(* Logix 5000 project; controller cal1615 1756-L62 rev 16.20; software revision 16.05; part 46 of 78 *)
(* tags used below, declared in another part *)
   FAULT : BOOL;   // Fault AFI
   HMI : BOOL;   // AFI HMI
   p01r02 : routine;   // System Misc Control
   p01r09_pb_global_reset : BOOL;   // System Modes PB: Global Fault Reset
   p01r09_stretch_mode : BOOL;
   p22_ai_amps : REAL;   // Tension Stand 1 Analog Input Tension Stand 1 Motor Current
   p22_ai_hz : REAL;   // Tension Stand 1 Analog Input Tension Stand 1 Motor Hertz
   p22_ai_speed : REAL;
   p22_ai_torque : REAL;
   p22_ai_ts1_lc : REAL;   // Tension Stand 1 Analog Input Loadcell
   p22_ao_selected_speed : REAL;   // Tension Stand 1 VFD Selected Speed
   p22_ao_torque : REAL;
   p22_ao_vfd : REAL;
   p22_control_word : INT;
   p22_di_brake : BOOL;   // Tension Stand 1 Digital Input Brake Temperature OK
   p22_di_close_nip_roll : BOOL;   // Tension Stand 1 Digital Input SS: Close Nip Roll
   p22_di_jog : BOOL;   // Tension Stand 1 Digital Input SS: Jog
   p22_di_jog_fwd : BOOL;   // Tension Stand 1 Digital Input PB: Jog Forward
   p22_di_jog_rev : BOOL;   // Tension Stand 1 Digital Input PB: Jog Reverse
   p22_di_open_nip_roll : BOOL;   // Tension Stand 1 Digital Input SS: Open Nip Roll
   p22_di_run : BOOL;   // Tension Stand 1 Digital Input SS: Run
   p22_di_therm : BOOL;   // Tension Stand 1 Digital Input Motor Temperature OK
   p22_dint_to_hmi : DINT[16];   // Tension Stand 1 Dint to HMI
   p22_do_close_nip_roll : BOOL;   // Tension Stand 1 Digital Output Close Tension Stand 1 Nip Roll
   p22_status_word : INT;
   p22_ts1_gear_ratio : REAL;
   p22_ts1_roll_diameter_ft : REAL;
   p22_vfd_input_max : REAL;
   p22_vfd_input_min : REAL;
   p22_vfd_output_max : REAL;
   p22_vfd_output_min : REAL;
   p22r01 : routine;   // Tension Stand 1 Main
   p22r03 : routine;   // Tension Stand 1 Input
   p22r03_ave_tq : REAL;
   p22r03_hz : SYS_SCP;   // Tension Stand 1 Analog Inputs SCP Hz
   p22r03_lc_input_max : REAL;
   p22r03_lc_input_min : REAL;
   p22r03_lc_output_max : REAL;
   p22r03_lc_output_min : REAL;
   p22r03_lc_scp : SYS_SCP;   // Tension Stand 1 Analog Input Load Cell Scaling
   p22r03_sample_timer : TIMER;
   p22r03_scaled_vfd_in : REAL;
   p22r03_timer_fault : TIMER[4];   // Tension Stand 1 Input Fault Delay
   p22r03_timer_warning : TIMER[4];   // Tension Stand 1 Input Warning Delay
   p22r03_tq_ave_ctrl : CONTROL;
   p22r03_tq_buffer : REAL[20];
   p22r03_tq_fifo : CONTROL;
   p22R03_ts1_vfd_rpm_to_speed : SYS_RPM_TO_SPEED;   // Tension Stand 1 Analog Input VFD RPM to Roll Surface Speed
   p22r03_unload : DINT;
   p22r03_vfd_in_scaling : SYS_SCP;
   p22r03_vfd_input_max : REAL;
   p22r03_vfd_input_min : REAL;
   p22r03_vfd_out_scaling : SYS_SCP;
   p22r03_vfd_output_max : REAL;
   p22r03_vfd_output_min : REAL;
   p22r04 : routine;   // Tension Stand 1 Output
   p22r04_speed_to_vfd_1 : SYS_SPEED_TO_VFD;   // Tension Stand 1 Analog Output Speed to VFD
   p22r04_timer_fault : TIMER[4];   // Tension Stand 1 Output Fault Delay
   p22r04_timer_warning : TIMER[4];   // Tension Stand 1 Output Warning Delay
   p22r05 : routine;   // Tension Stand 1 Dint to HMI
   p22r05_timer_fault : TIMER[4];   // Tension Stand 1 Dint to HMI Fault Delay
   p22r05_timer_warning : TIMER[4];   // Tension Stand 1 Dint to HMI Warning Delay
   p22r09_mode_jog : BOOL;   // Tension Stand 1 Modes Jog Mode
   p22r09_mode_run : BOOL;   // Tension Stand 1 Modes Run Mode
   p22r09_mode_thread : BOOL;   // Tension Stand 1 Modes Thread Mode
   p25r03 : routine;
(* P22_Tension_Stand_1, continued *)

ROUTINE R03_Input   (* ladder *)
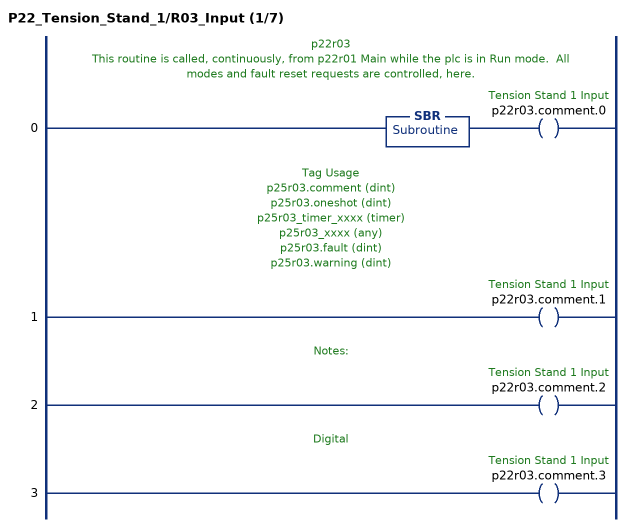
   // p22r03
   // This routine is called, continuously, from p22r01 Main while the plc is in Run mode.  All modes and fault reset requests are controlled, here.
   0: SBR()OTE(p22r03.comment.0);
   // Tag Usage
   // p25r03.comment (dint)
   // p25r03.oneshot (dint)
   // p25r03_timer_xxxx (timer)
   // p25r03_xxxx (any)
   // p25r03.fault (dint)
   // p25r03.warning (dint)
   1: OTE(p22r03.comment.1);
   // Notes:
   2: OTE(p22r03.comment.2);
   // Digital
   3: OTE(p22r03.comment.3);
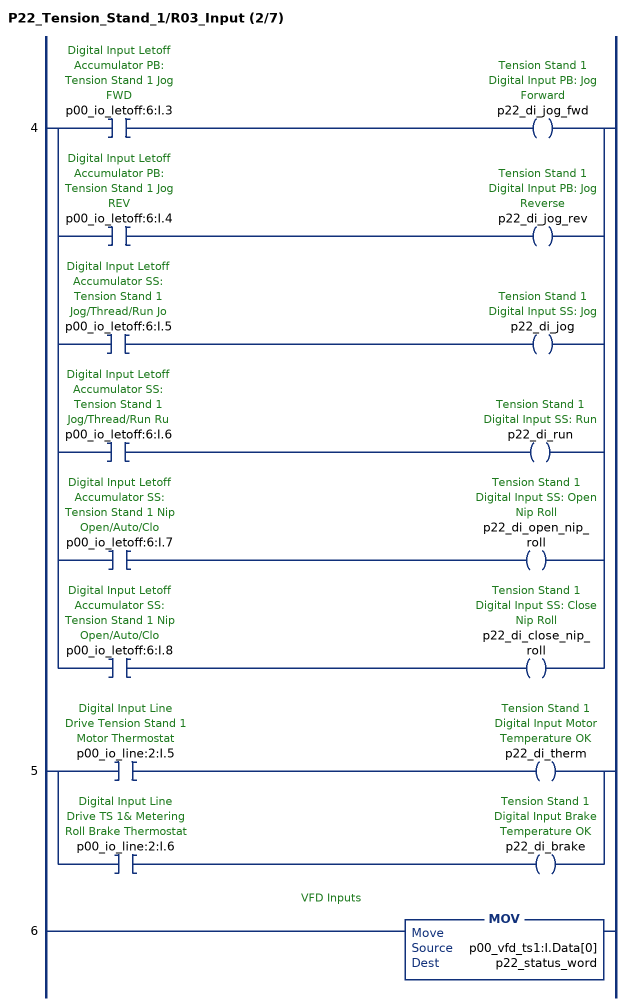
   4: [XIC(p00_io_letoff:6:I.3) OTE(p22_di_jog_fwd) ,XIC(p00_io_letoff:6:I.4) OTE(p22_di_jog_rev) ,XIC(p00_io_letoff:6:I.5) OTE(p22_di_jog) ,XIC(p00_io_letoff:6:I.6) OTE(p22_di_run) ,XIC(p00_io_letoff:6:I.7) OTE(p22_di_open_nip_roll) ,XIC(p00_io_letoff:6:I.8) OTE(p22_di_close_nip_roll) ];
   5: [XIC(p00_io_line:2:I.5) OTE(p22_di_therm) ,XIC(p00_io_line:2:I.6) OTE(p22_di_brake) ];
   // VFD Inputs
   6: MOV(p00_vfd_ts1:I.Data[0],p22_status_word);
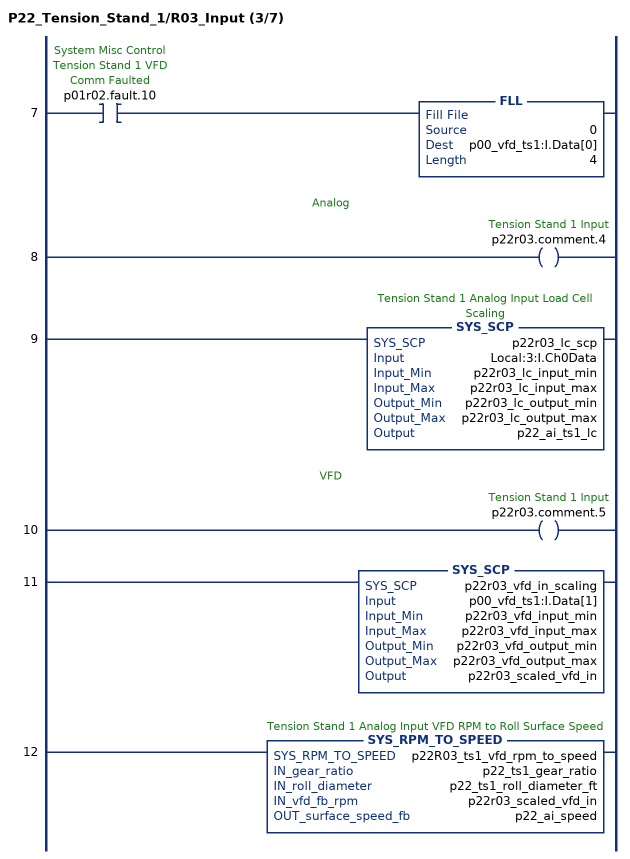
   7: XIC(p01r02.fault.10)FLL(0,p00_vfd_ts1:I.Data[0],4);
   // Analog
   8: OTE(p22r03.comment.4);
   9: SYS_SCP(p22r03_lc_scp,Local:3:I.Ch0Data,p22r03_lc_input_min,p22r03_lc_input_max,p22r03_lc_output_min,p22r03_lc_output_max,p22_ai_ts1_lc);
   // VFD
   10: OTE(p22r03.comment.5);
   11: SYS_SCP(p22r03_vfd_in_scaling,p00_vfd_ts1:I.Data[1],p22r03_vfd_input_min,p22r03_vfd_input_max,p22r03_vfd_output_min,p22r03_vfd_output_max,p22r03_scaled_vfd_in);
   12: SYS_RPM_TO_SPEED(p22R03_ts1_vfd_rpm_to_speed,p22_ts1_gear_ratio,p22_ts1_roll_diameter_ft,p22r03_scaled_vfd_in,p22_ai_speed);
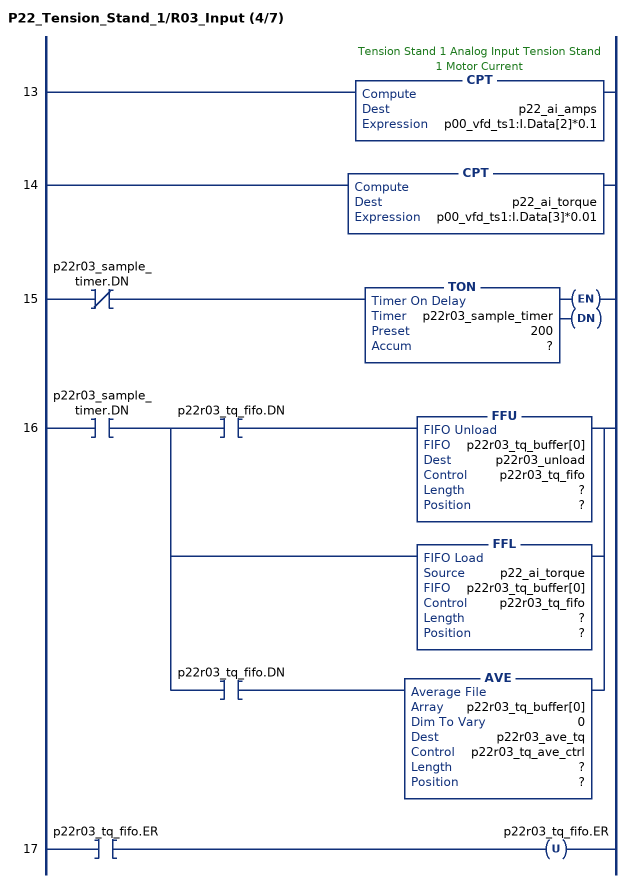
   13: CPT(p22_ai_amps,p00_vfd_ts1:I.Data[2]*0.1);
   14: CPT(p22_ai_torque,p00_vfd_ts1:I.Data[3]*0.01);
   15: XIO(p22r03_sample_timer.DN)TON(p22r03_sample_timer,?,?);
   16: XIC(p22r03_sample_timer.DN)[XIC(p22r03_tq_fifo.DN) FFU(p22r03_tq_buffer[0],p22r03_unload,p22r03_tq_fifo,?,?) ,FFL(p22_ai_torque,p22r03_tq_buffer[0],p22r03_tq_fifo,?,?) ,XIC(p22r03_tq_fifo.DN) AVE(p22r03_tq_buffer[0],0,p22r03_ave_tq,p22r03_tq_ave_ctrl,?,?) ];
   17: XIC(p22r03_tq_fifo.ER)OTU(p22r03_tq_fifo.ER);
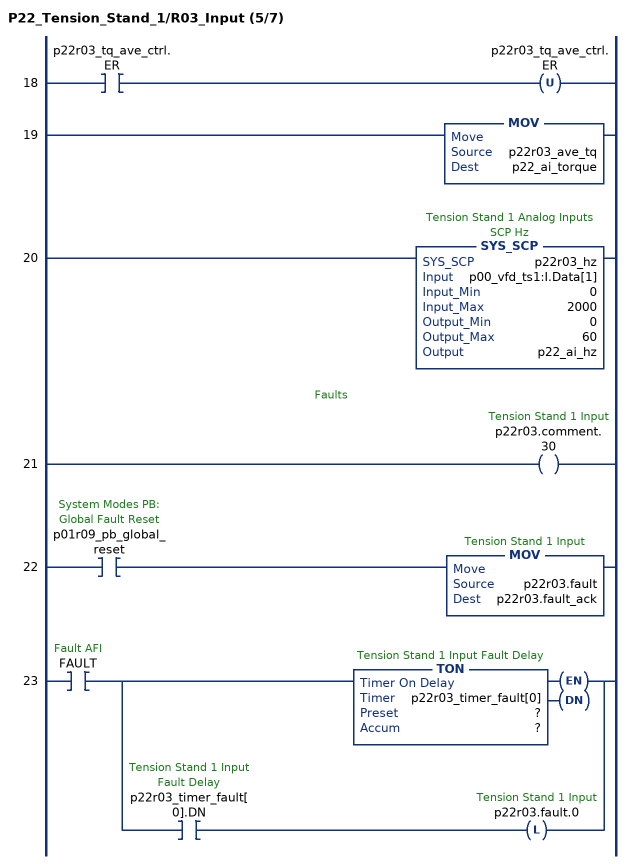
   18: XIC(p22r03_tq_ave_ctrl.ER)OTU(p22r03_tq_ave_ctrl.ER);
   19: MOV(p22r03_ave_tq,p22_ai_torque);
   20: SYS_SCP(p22r03_hz,p00_vfd_ts1:I.Data[1],0,2000,0,60,p22_ai_hz);
   // Faults
   21: OTE(p22r03.comment.30);
   22: XIC(p01r09_pb_global_reset)MOV(p22r03.fault,p22r03.fault_ack);
   23: XIC(FAULT)[TON(p22r03_timer_fault[0],?,?) ,XIC(p22r03_timer_fault[0].DN) OTL(p22r03.fault.0) ];
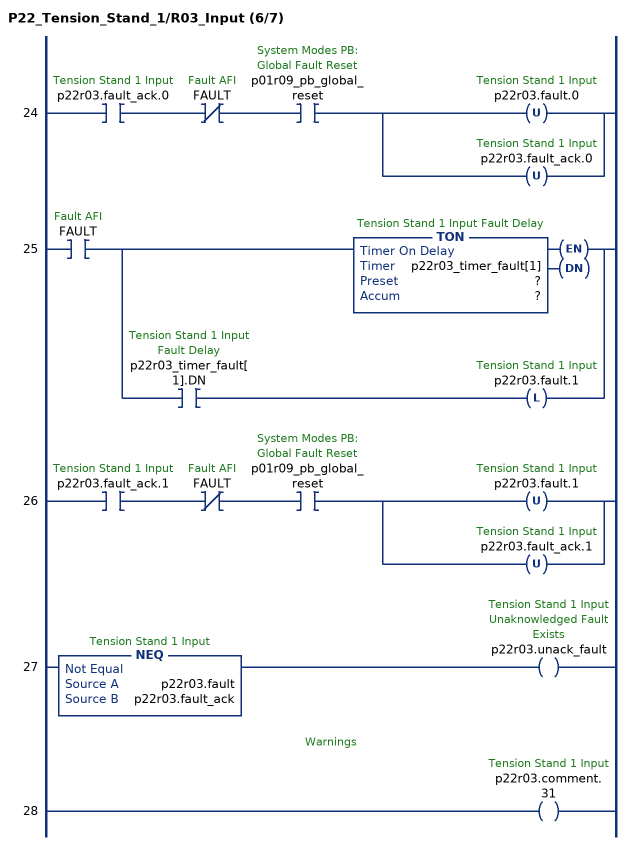
   24: XIC(p22r03.fault_ack.0)XIO(FAULT)XIC(p01r09_pb_global_reset)[OTU(p22r03.fault.0) ,OTU(p22r03.fault_ack.0) ];
   25: XIC(FAULT)[TON(p22r03_timer_fault[1],?,?) ,XIC(p22r03_timer_fault[1].DN) OTL(p22r03.fault.1) ];
   26: XIC(p22r03.fault_ack.1)XIO(FAULT)XIC(p01r09_pb_global_reset)[OTU(p22r03.fault.1) ,OTU(p22r03.fault_ack.1) ];
   27: NEQ(p22r03.fault,p22r03.fault_ack)OTE(p22r03.unack_fault);
   // Warnings
   28: OTE(p22r03.comment.31);
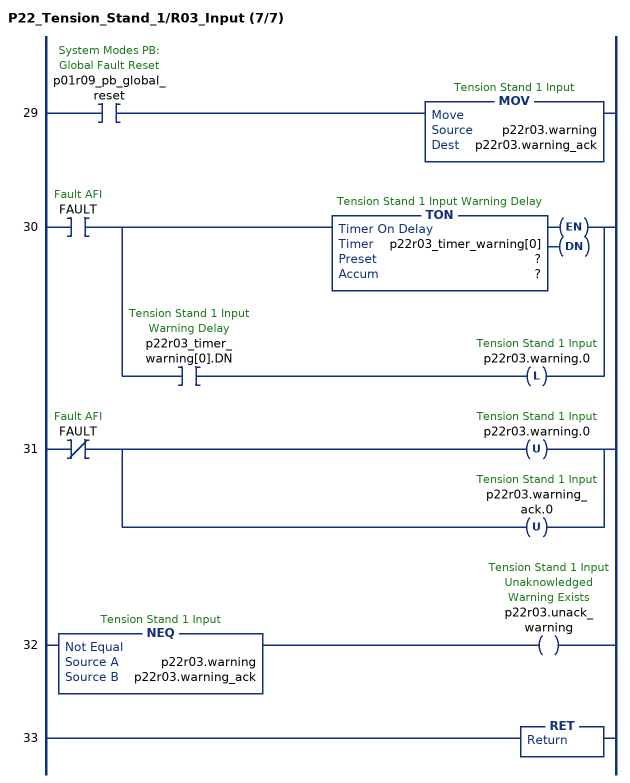
   29: XIC(p01r09_pb_global_reset)MOV(p22r03.warning,p22r03.warning_ack);
   30: XIC(FAULT)[TON(p22r03_timer_warning[0],?,?) ,XIC(p22r03_timer_warning[0].DN) OTL(p22r03.warning.0) ];
   31: XIO(FAULT)[OTU(p22r03.warning.0) ,OTU(p22r03.warning_ack.0) ];
   32: NEQ(p22r03.warning,p22r03.warning_ack)OTE(p22r03.unack_warning);
   33: RET();
END_ROUTINE

ROUTINE R04_Output   (* ladder *)
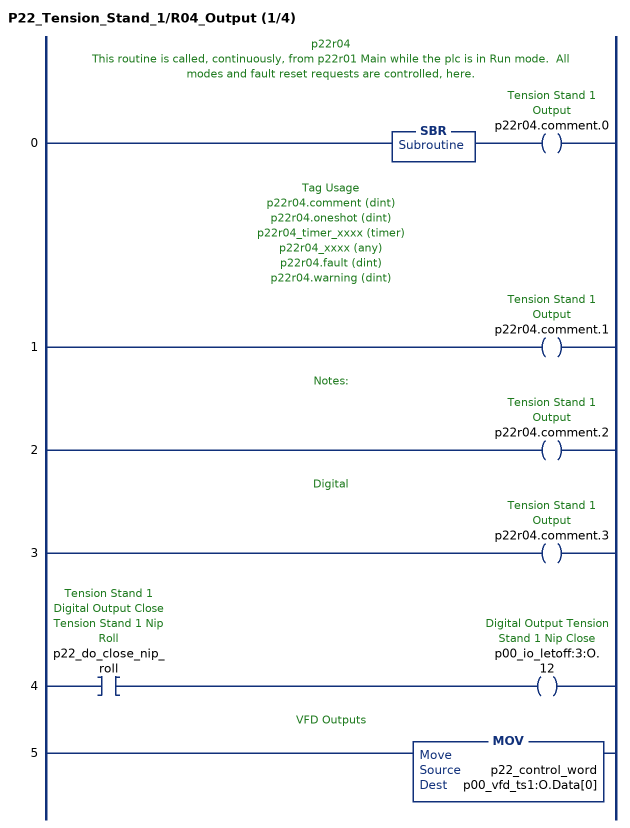
   // p22r04
   // This routine is called, continuously, from p22r01 Main while the plc is in Run mode.  All modes and fault reset requests are controlled, here.
   0: SBR()OTE(p22r04.comment.0);
   // Tag Usage
   // p22r04.comment (dint)
   // p22r04.oneshot (dint)
   // p22r04_timer_xxxx (timer)
   // p22r04_xxxx (any)
   // p22r04.fault (dint)
   // p22r04.warning (dint)
   1: OTE(p22r04.comment.1);
   // Notes:
   2: OTE(p22r04.comment.2);
   // Digital
   3: OTE(p22r04.comment.3);
   4: XIC(p22_do_close_nip_roll)OTE(p00_io_letoff:3:O.12);
   // VFD Outputs
   5: MOV(p22_control_word,p00_vfd_ts1:O.Data[0]);
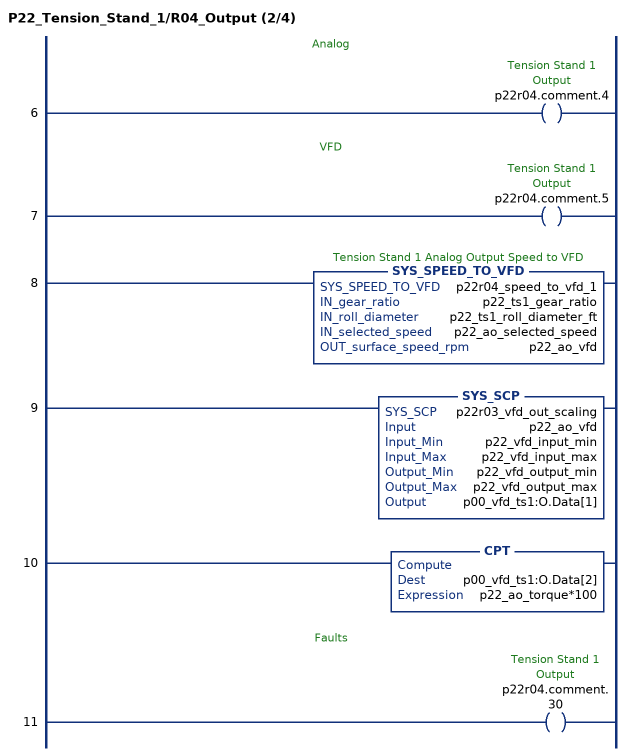
   // Analog
   6: OTE(p22r04.comment.4);
   // VFD
   7: OTE(p22r04.comment.5);
   8: SYS_SPEED_TO_VFD(p22r04_speed_to_vfd_1,p22_ts1_gear_ratio,p22_ts1_roll_diameter_ft,p22_ao_selected_speed,p22_ao_vfd);
   9: SYS_SCP(p22r03_vfd_out_scaling,p22_ao_vfd,p22_vfd_input_min,p22_vfd_input_max,p22_vfd_output_min,p22_vfd_output_max,p00_vfd_ts1:O.Data[1]);
   10: CPT(p00_vfd_ts1:O.Data[2],p22_ao_torque*100);
   // Faults
   11: OTE(p22r04.comment.30);
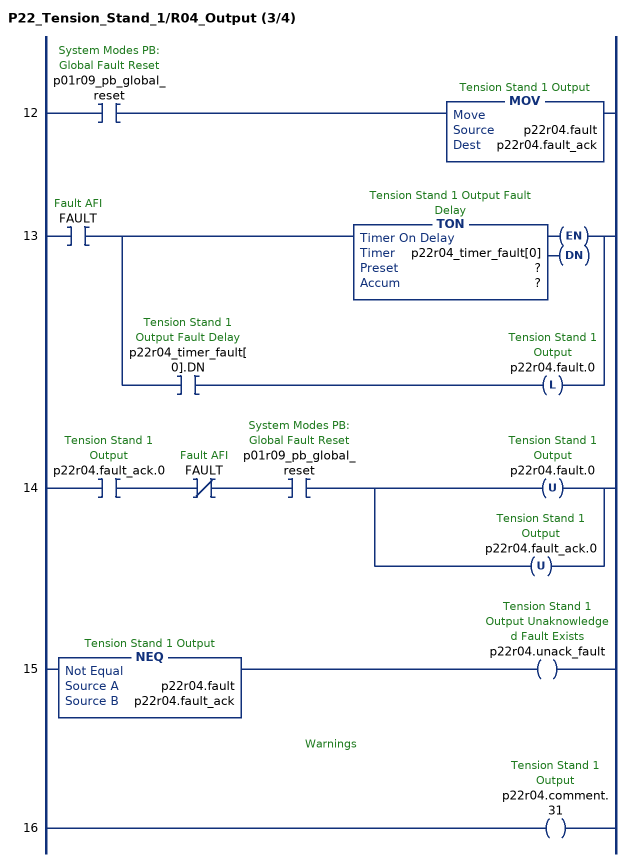
   12: XIC(p01r09_pb_global_reset)MOV(p22r04.fault,p22r04.fault_ack);
   13: XIC(FAULT)[TON(p22r04_timer_fault[0],?,?) ,XIC(p22r04_timer_fault[0].DN) OTL(p22r04.fault.0) ];
   14: XIC(p22r04.fault_ack.0)XIO(FAULT)XIC(p01r09_pb_global_reset)[OTU(p22r04.fault.0) ,OTU(p22r04.fault_ack.0) ];
   15: NEQ(p22r04.fault,p22r04.fault_ack)OTE(p22r04.unack_fault);
   // Warnings
   16: OTE(p22r04.comment.31);
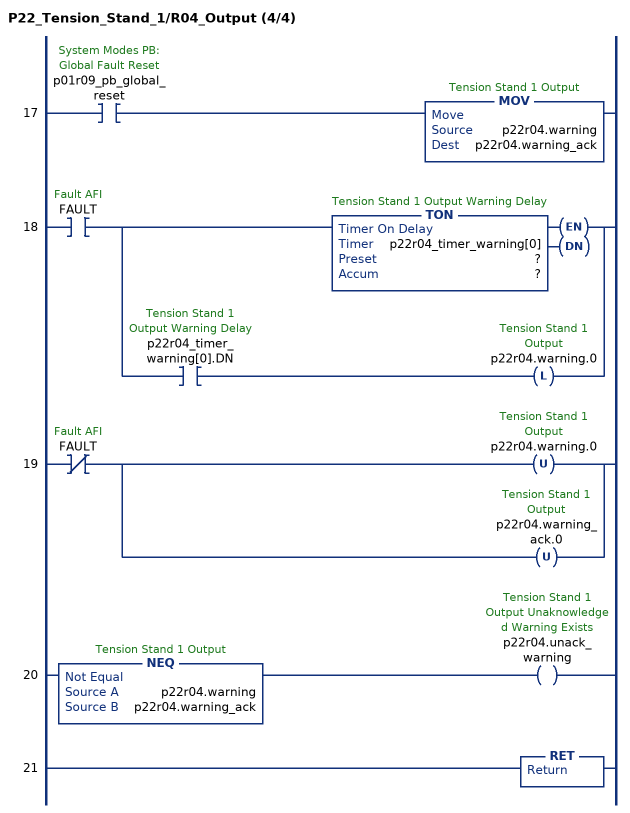
   17: XIC(p01r09_pb_global_reset)MOV(p22r04.warning,p22r04.warning_ack);
   18: XIC(FAULT)[TON(p22r04_timer_warning[0],?,?) ,XIC(p22r04_timer_warning[0].DN) OTL(p22r04.warning.0) ];
   19: XIO(FAULT)[OTU(p22r04.warning.0) ,OTU(p22r04.warning_ack.0) ];
   20: NEQ(p22r04.warning,p22r04.warning_ack)OTE(p22r04.unack_warning);
   21: RET();
END_ROUTINE

ROUTINE R05_Dint_to_HMI   (* ladder *)
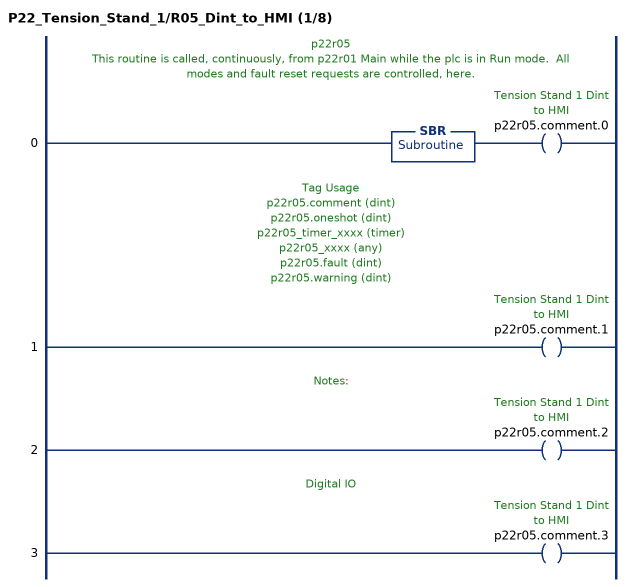
   // p22r05
   // This routine is called, continuously, from p22r01 Main while the plc is in Run mode.  All modes and fault reset requests are controlled, here.
   0: SBR()OTE(p22r05.comment.0);
   // Tag Usage
   // p22r05.comment (dint)
   // p22r05.oneshot (dint)
   // p22r05_timer_xxxx (timer)
   // p22r05_xxxx (any)
   // p22r05.fault (dint)
   // p22r05.warning (dint)
   1: OTE(p22r05.comment.1);
   // Notes:
   2: OTE(p22r05.comment.2);
   // Digital IO
   3: OTE(p22r05.comment.3);
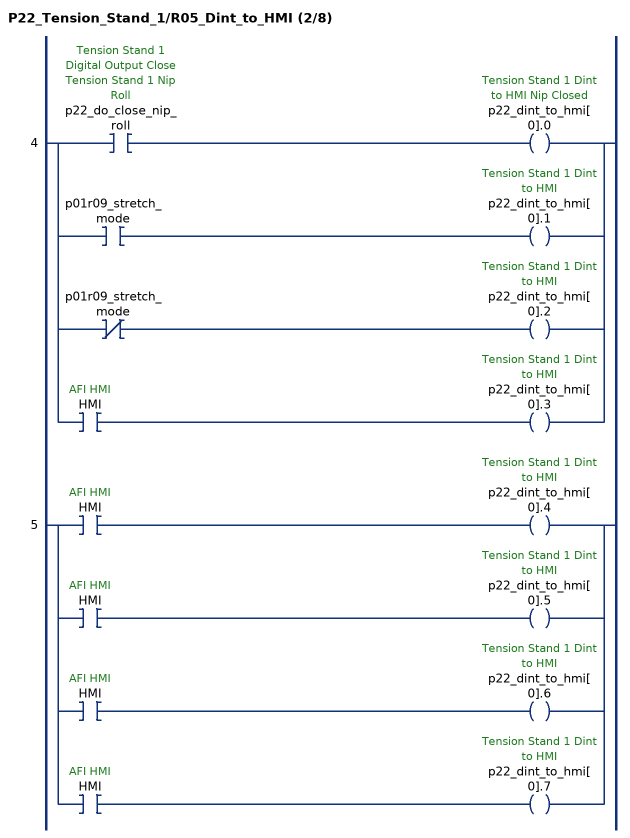
   4: [XIC(p22_do_close_nip_roll) OTE(p22_dint_to_hmi[0].0) ,XIC(p01r09_stretch_mode) OTE(p22_dint_to_hmi[0].1) ,XIO(p01r09_stretch_mode) OTE(p22_dint_to_hmi[0].2) ,XIC(HMI) OTE(p22_dint_to_hmi[0].3) ];
   5: [XIC(HMI) OTE(p22_dint_to_hmi[0].4) ,XIC(HMI) OTE(p22_dint_to_hmi[0].5) ,XIC(HMI) OTE(p22_dint_to_hmi[0].6) ,XIC(HMI) OTE(p22_dint_to_hmi[0].7) ];
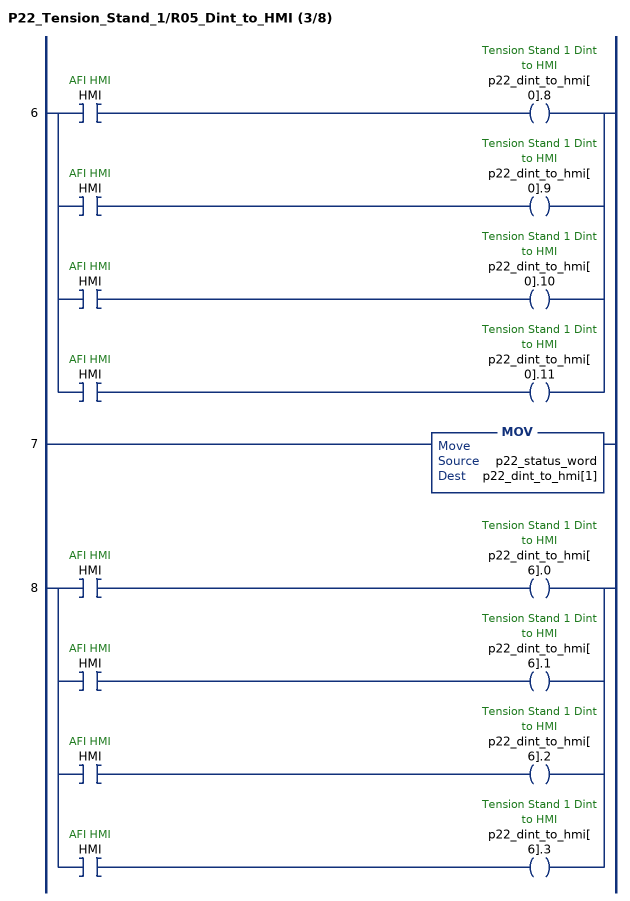
   6: [XIC(HMI) OTE(p22_dint_to_hmi[0].8) ,XIC(HMI) OTE(p22_dint_to_hmi[0].9) ,XIC(HMI) OTE(p22_dint_to_hmi[0].10) ,XIC(HMI) OTE(p22_dint_to_hmi[0].11) ];
   7: MOV(p22_status_word,p22_dint_to_hmi[1]);
   8: [XIC(HMI) OTE(p22_dint_to_hmi[6].0) ,XIC(HMI) OTE(p22_dint_to_hmi[6].1) ,XIC(HMI) OTE(p22_dint_to_hmi[6].2) ,XIC(HMI) OTE(p22_dint_to_hmi[6].3) ];
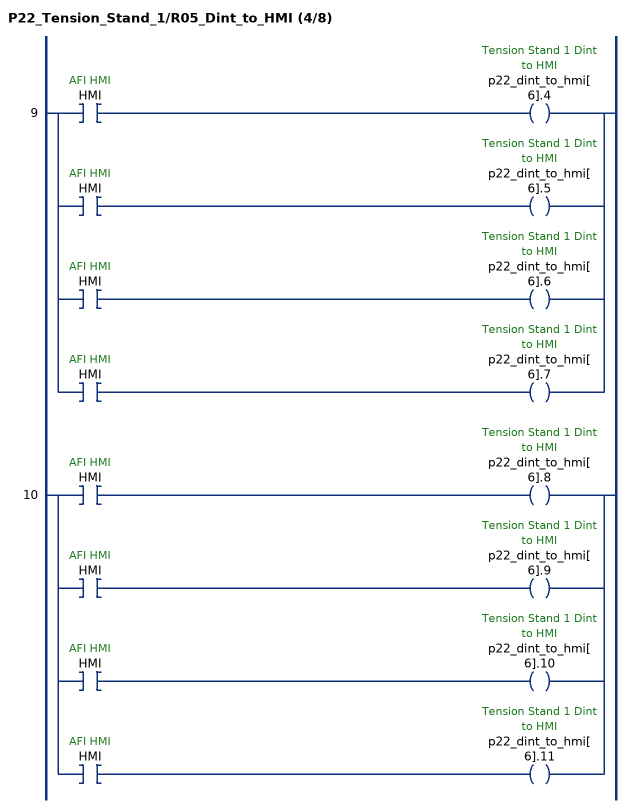
   9: [XIC(HMI) OTE(p22_dint_to_hmi[6].4) ,XIC(HMI) OTE(p22_dint_to_hmi[6].5) ,XIC(HMI) OTE(p22_dint_to_hmi[6].6) ,XIC(HMI) OTE(p22_dint_to_hmi[6].7) ];
   10: [XIC(HMI) OTE(p22_dint_to_hmi[6].8) ,XIC(HMI) OTE(p22_dint_to_hmi[6].9) ,XIC(HMI) OTE(p22_dint_to_hmi[6].10) ,XIC(HMI) OTE(p22_dint_to_hmi[6].11) ];
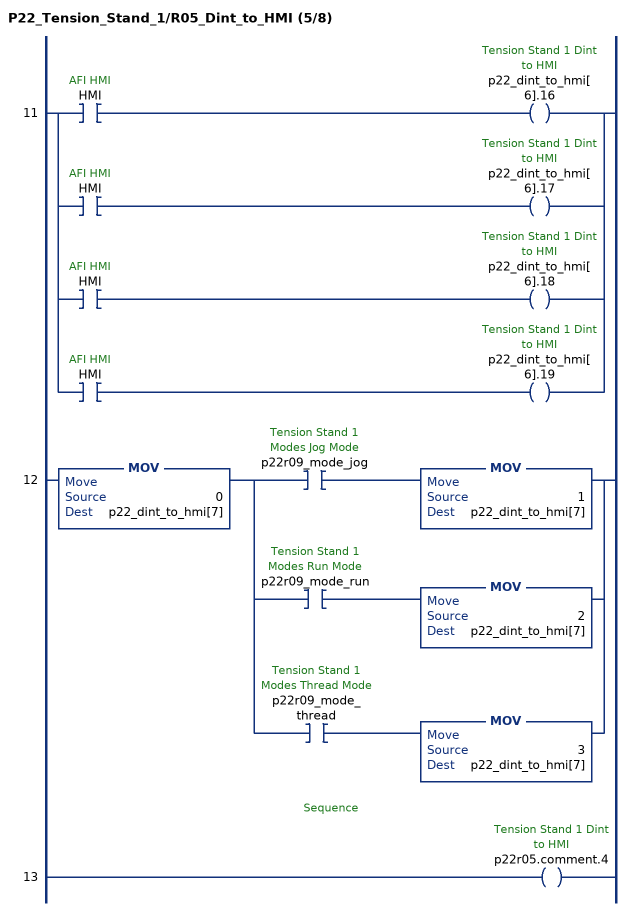
   11: [XIC(HMI) OTE(p22_dint_to_hmi[6].16) ,XIC(HMI) OTE(p22_dint_to_hmi[6].17) ,XIC(HMI) OTE(p22_dint_to_hmi[6].18) ,XIC(HMI) OTE(p22_dint_to_hmi[6].19) ];
   12: MOV(0,p22_dint_to_hmi[7])[XIC(p22r09_mode_jog) MOV(1,p22_dint_to_hmi[7]) ,XIC(p22r09_mode_run) MOV(2,p22_dint_to_hmi[7]) ,XIC(p22r09_mode_thread) MOV(3,p22_dint_to_hmi[7]) ];
   // Sequence
   13: OTE(p22r05.comment.4);
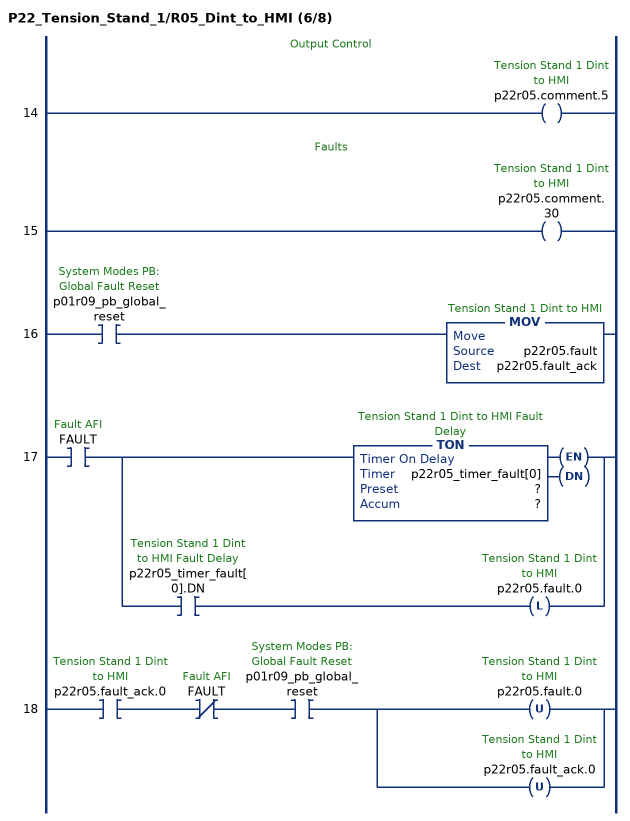
   // Output Control
   14: OTE(p22r05.comment.5);
   // Faults
   15: OTE(p22r05.comment.30);
   16: XIC(p01r09_pb_global_reset)MOV(p22r05.fault,p22r05.fault_ack);
   17: XIC(FAULT)[TON(p22r05_timer_fault[0],?,?) ,XIC(p22r05_timer_fault[0].DN) OTL(p22r05.fault.0) ];
   18: XIC(p22r05.fault_ack.0)XIO(FAULT)XIC(p01r09_pb_global_reset)[OTU(p22r05.fault.0) ,OTU(p22r05.fault_ack.0) ];
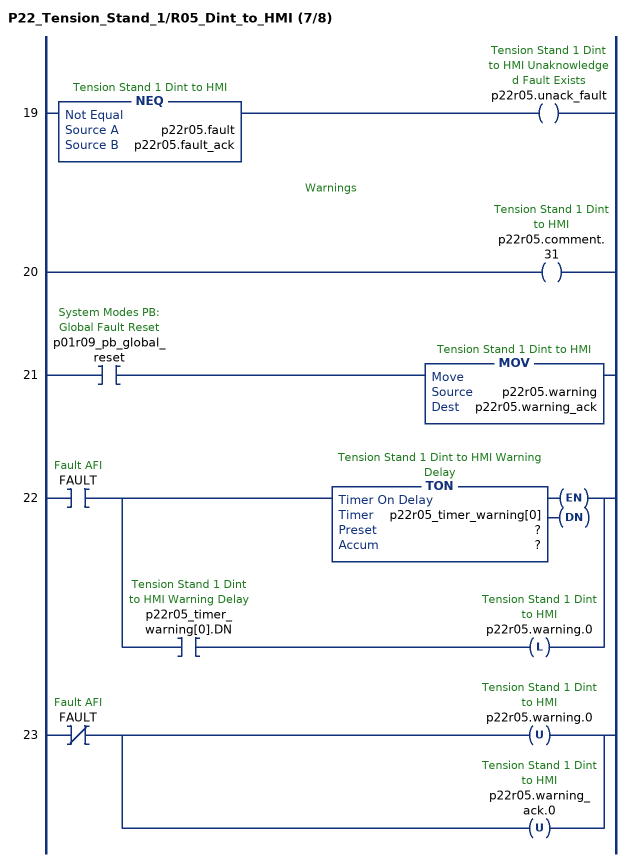
   19: NEQ(p22r05.fault,p22r05.fault_ack)OTE(p22r05.unack_fault);
   // Warnings
   20: OTE(p22r05.comment.31);
   21: XIC(p01r09_pb_global_reset)MOV(p22r05.warning,p22r05.warning_ack);
   22: XIC(FAULT)[TON(p22r05_timer_warning[0],?,?) ,XIC(p22r05_timer_warning[0].DN) OTL(p22r05.warning.0) ];
   23: XIO(FAULT)[OTU(p22r05.warning.0) ,OTU(p22r05.warning_ack.0) ];
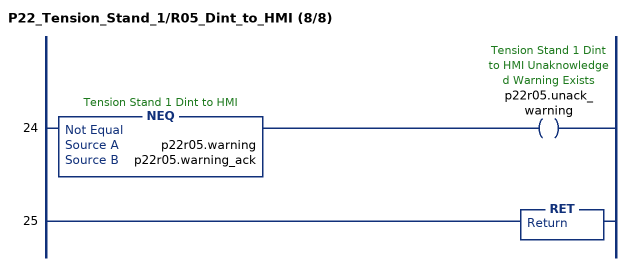
   24: NEQ(p22r05.warning,p22r05.warning_ack)OTE(p22r05.unack_warning);
   25: RET();
END_ROUTINE
